Staubli VAL3: onF7Event.pgx

program onF7Event()
  local num l_nItem
begin

end
